Omron CX-Programmer project 新工程 (CX-Programmer 9.61)

# PLC 新PLC1: CP1E N30

## Global symbols (name address type ; comment)
0.00 BOOL  ; 启动开关
0.01 BOOL  ; 切换开关
100.00 BOOL  ; 绿灯1
100.02 BOOL  ; 红灯1
100.03 BOOL  ; 红灯2
100.04 BOOL  ; 绿灯2
100.05 BOOL  ; 黄灯2

## Program 新程序1 (cyclic task 0)

### Section 段1

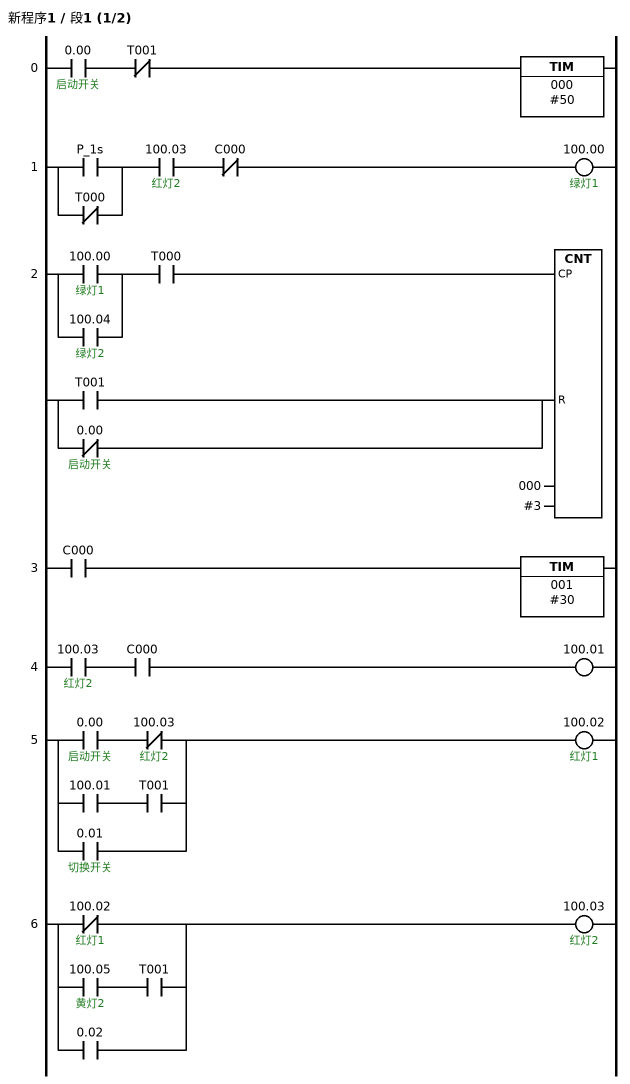
; rung 0
LD 0.00  ; 启动开关
ANDNOT T001
TIM 000 #50
; rung 1
LD P_1s
ORNOT T000
AND 100.03  ; 红灯2
ANDNOT C000
OUT 100.00  ; 绿灯1
; rung 2
LD 100.00  ; 绿灯1
OR 100.04  ; 绿灯2
AND T000
LD T001
ORNOT 0.00  ; 启动开关
CNT 000 #3
; rung 3
LD C000
TIM 001 #30
; rung 4
LD 100.03  ; 红灯2
AND C000
OUT 100.01
; rung 5
LD 0.00  ; 启动开关
ANDNOT 100.03  ; 红灯2
LD 100.01
AND T001
ORLD
OR 0.01  ; 切换开关
OUT 100.02  ; 红灯1
; rung 6
LDNOT 100.02  ; 红灯1
LD 100.05  ; 黄灯2
AND T001
ORLD
OR 0.02
OUT 100.03  ; 红灯2

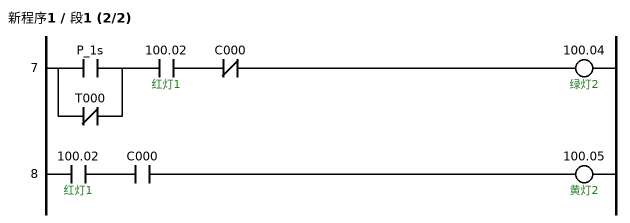
; rung 7
LD P_1s
ORNOT T000
AND 100.02  ; 红灯1
ANDNOT C000
OUT 100.04  ; 绿灯2
; rung 8
LD 100.02  ; 红灯1
AND C000
OUT 100.05  ; 黄灯2
; rung 9
END(001)

### Section END
; rung 0
END(001)